FUNCTION Rotation : INT
VAR_INPUT
	EndPosition: INT;
	State: INT;
END_VAR
VAR
	MovementEnum: Movement;
	NextState: INT;
	MotorDirectionEnum: MovementDirection;
END_VAR

IF Automatic.RotationPositionAuto > EndPosition THEN
	MotorDirectionEnum := MovementDirection.TowardsSensor;
ELSE
	MotorDirectionEnum := MovementDirection.AwayFromSensor;
END_IF

IF MotorDirectionEnum = MovementDirection.TowardsSensor THEN
	IF Automatic.RotationPositionAuto > EndPosition THEN
		IO.MotorRotationDirection := (MotorDirectionEnum = MovementDirection.TowardsSensor);
		IF NOT Automatic.SafetyRON THEN
			Automatic.RCurrentlyMoving := TRUE;
			IO.MotorRotation := (MovementEnum = Movement.ON);
		END_IF
		NextState := State;
	ELSE
		IO.MotorRotation := (MovementEnum = Movement.OFF);
		NextState := State + 1;
		Automatic.RCurrentlyMoving := FALSE;
	END_IF
ELSE
	IF Automatic.RotationPositionAuto < EndPosition THEN
		IO.MotorRotationDirection := (MotorDirectionEnum = MovementDirection.AwayFromSensor);
		IF NOT Automatic.SafetyRON THEN
			Automatic.RCurrentlyMoving := TRUE;
			IO.MotorRotation := (MovementEnum = Movement.ON);
		END_IF
		NextState := State;
	ELSE
		IO.MotorRotation := (MovementEnum = Movement.OFF);
		NextState := State + 1;
		Automatic.RCurrentlyMoving := FALSE;
	END_IF
END_IF

Rotation := NextState;
RETURN;

END_FUNCTION

(* stored: Version 1.1.0.1, ProductVersion 3.1.4024.13
   POU Rotation: Id {b022b9d3-a89d-42d2-9989-464d993048d9}, SpecialFunc None *)
